(* Schneider Machine Expert - Basic project DDEF, file version 2.7.0.0 *)
(* ProjectInformations: Name=Novo projeto *)

HARDWARE
  Cpu 0: TM221CE24R
  EthernetConfiguration: NetworkName=M221, IpAllocationMode=FixedAddress, IpAddress=0.0.0.0, SubnetMask=0.0.0.0
  SerialLineConfiguration: Baud=Baud19200, Parity=ParityEven, DataBits=DataBits8, StopBits=StopBits1, PhysicalMedium=PhysicalMediumRs485, TransmissionMode=TransmissionModeModbusRtu, SlaveId=1, Addressing=SlaveAddressing
  MastTask: UsePeriodScanMode=false, PeriodScan=100
  FastTask: Period=255
  CpuBehavior: StartingMode=StartAsPreviousState, AutoSaveRamOnEeprom=true, WatchdogPeriod=250

SYMBOLS  (address, symbol, comment, settings)
  %M0       START_
  %M1       STOP
  %M2       RESET
  %M3       EMERGENCIA
  %M4       MANUAL
  %M5       AUTO
  %M6       L_START
  %M7       L_RESET
  %M8       L_STOP
  %M9       L_MANUAL
  %M10      L_AUTO
  %MW0      SNIVEL
  %MW1      SETPOINT
  %MW2      V_ENCHE
  %MW3      V_DESCARGA
  %MW4      V_SETPOINT
  %MW5      V_NIVEL

POU Novo POU
  (* SectionNumber=1 *)

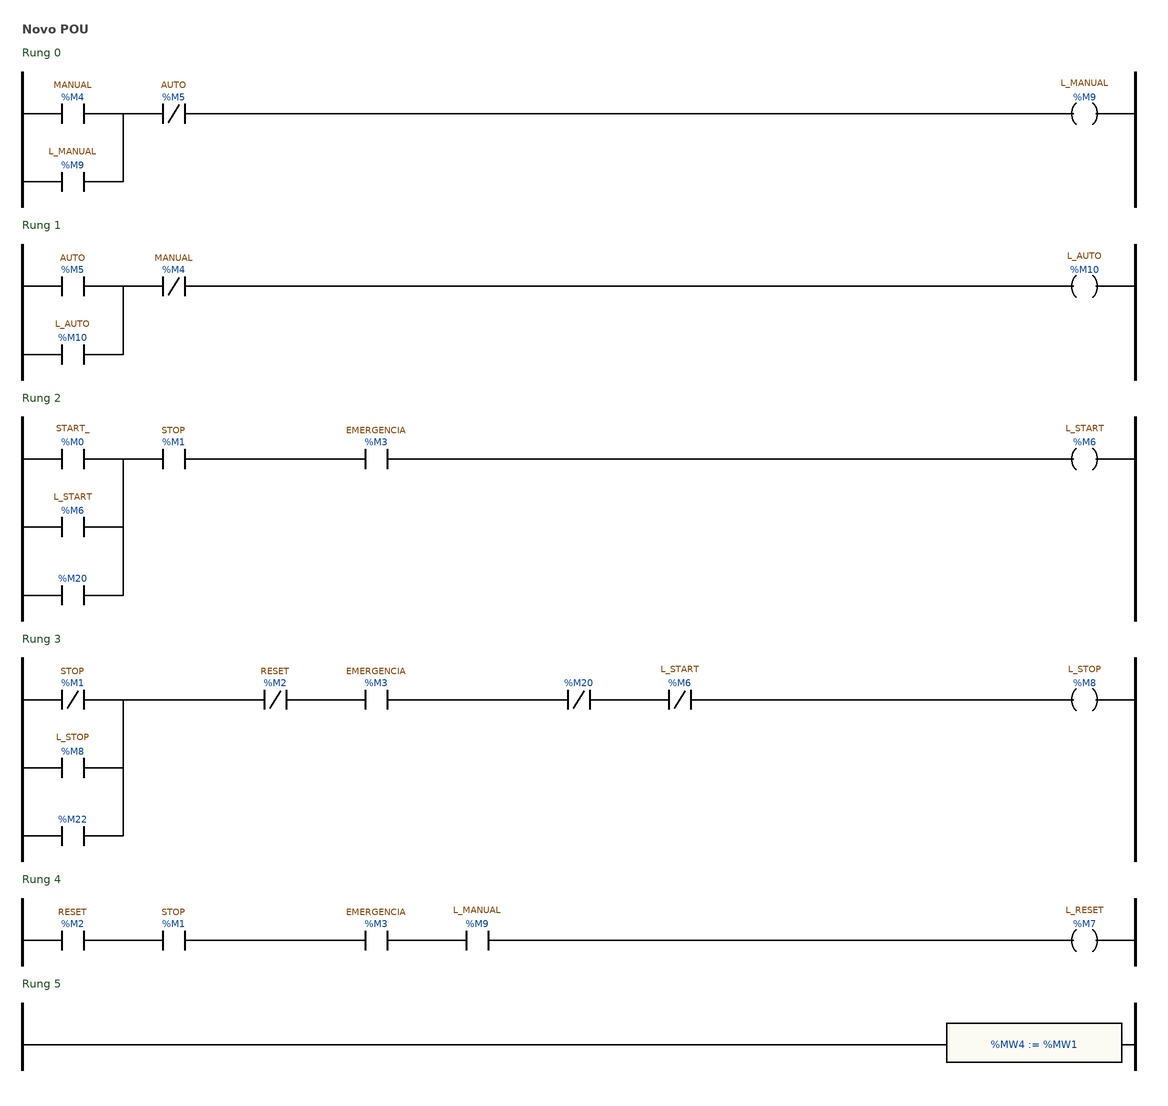

// Rung 0
  LD %M4                  (* MANUAL *)
  OR %M9                  (* L_MANUAL *)
  ANDN %M5                (* AUTO *)
  ST %M9                  (* L_MANUAL *)
  // as ST:
  //   L_MANUAL := (MANUAL OR L_MANUAL) AND NOT AUTO;

// Rung 1
  LD %M5                  (* AUTO *)
  OR %M10                 (* L_AUTO *)
  ANDN %M4                (* MANUAL *)
  ST %M10                 (* L_AUTO *)
  // as ST:
  //   L_AUTO := (AUTO OR L_AUTO) AND NOT MANUAL;

// Rung 2
  LD %M0                  (* START_ *)
  OR %M6                  (* L_START *)
  OR %M20
  AND %M1                 (* STOP *)
  AND %M3                 (* EMERGENCIA *)
  ST %M6                  (* L_START *)
  // as ST:
  //   L_START := (START_ OR L_START OR %M20) AND STOP AND EMERGENCIA;

// Rung 3
  LDN %M1                 (* STOP *)
  OR %M8                  (* L_STOP *)
  OR %M22
  ANDN %M2                (* RESET *)
  AND %M3                 (* EMERGENCIA *)
  ANDN %M20
  ANDN %M6                (* L_START *)
  ST %M8                  (* L_STOP *)
  // as ST:
  //   L_STOP := (NOT STOP OR L_STOP OR %M22) AND NOT RESET AND EMERGENCIA AND NOT %M20 AND NOT L_START;

// Rung 4
  LD %M2                  (* RESET *)
  AND %M1                 (* STOP *)
  AND %M3                 (* EMERGENCIA *)
  AND %M9                 (* L_MANUAL *)
  ST %M7                  (* L_RESET *)
  // as ST:
  //   L_RESET := RESET AND STOP AND EMERGENCIA AND L_MANUAL;

// Rung 5
  LD 1
  [ %MW4 := %MW1 ]        (* V_SETPOINT, SETPOINT *)
  // as ST:
  //   V_SETPOINT := SETPOINT;

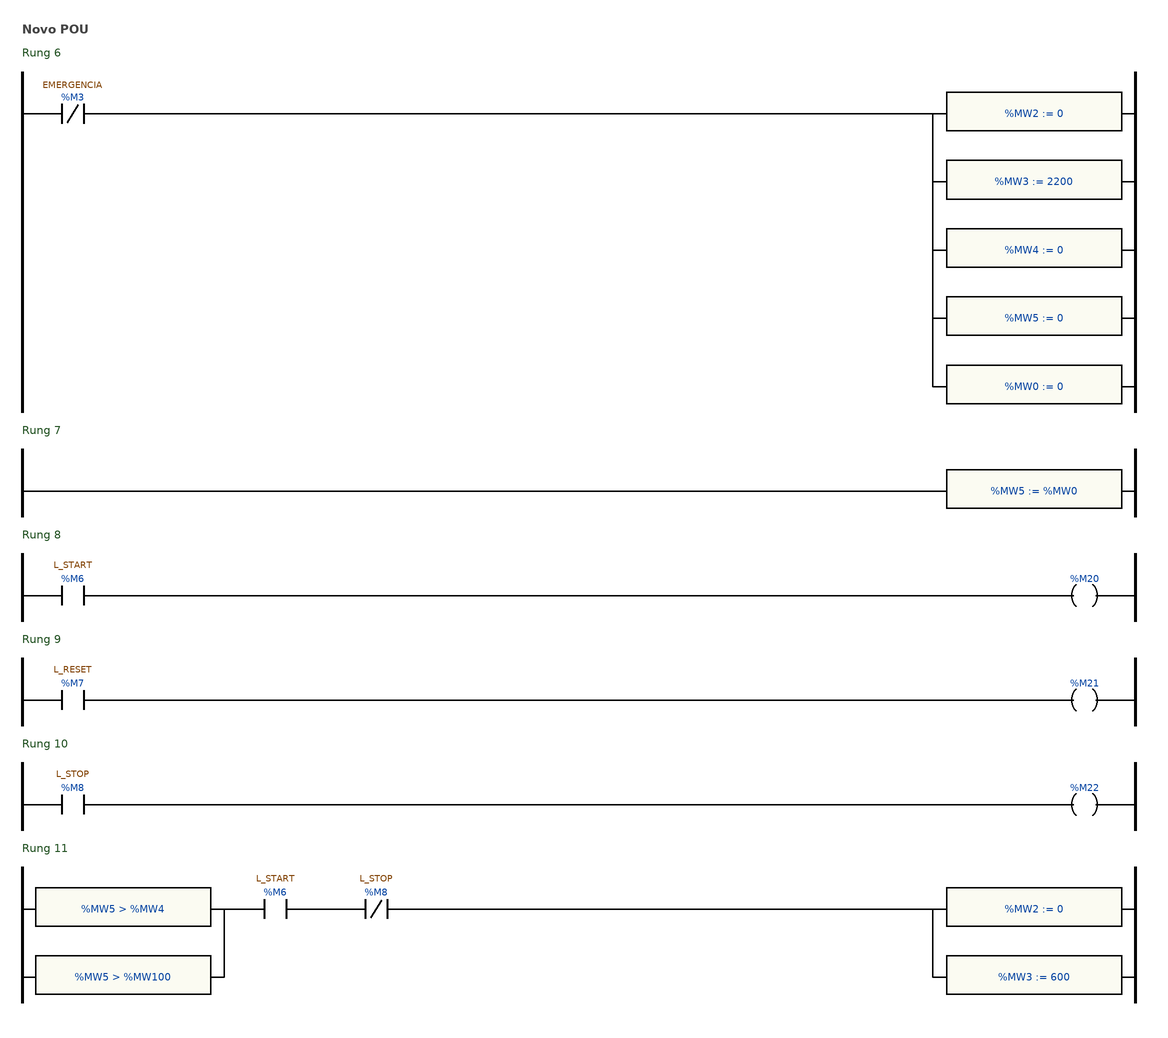

// Rung 6
  LDN %M3                 (* EMERGENCIA *)
  [ %MW2 := 0 ]           (* V_ENCHE *)
  [ %MW3 := 2200 ]        (* V_DESCARGA *)
  [ %MW4 := 0 ]           (* V_SETPOINT *)
  [ %MW5 := 0 ]           (* V_NIVEL *)
  [ %MW0 := 0 ]           (* SNIVEL *)
  // as ST:
  //   IF NOT EMERGENCIA THEN V_ENCHE := 0; END_IF;
  //   IF NOT EMERGENCIA THEN V_DESCARGA := 2200; END_IF;
  //   IF NOT EMERGENCIA THEN V_SETPOINT := 0; END_IF;
  //   IF NOT EMERGENCIA THEN V_NIVEL := 0; END_IF;
  //   IF NOT EMERGENCIA THEN SNIVEL := 0; END_IF;

// Rung 7
  LD 1
  [ %MW5 := %MW0 ]        (* V_NIVEL, SNIVEL *)
  // as ST:
  //   V_NIVEL := SNIVEL;

// Rung 8
  LD %M6                  (* L_START *)
  ST %M20
  // as ST:
  //   %M20 := L_START;

// Rung 9
  LD %M7                  (* L_RESET *)
  ST %M21
  // as ST:
  //   %M21 := L_RESET;

// Rung 10
  LD %M8                  (* L_STOP *)
  ST %M22
  // as ST:
  //   %M22 := L_STOP;

// Rung 11
  LD [ %MW5 > %MW4 ]      (* V_NIVEL, V_SETPOINT *)
  OR [ %MW5 > %MW100 ]    (* V_NIVEL *)
  AND %M6                 (* L_START *)
  ANDN %M8                (* L_STOP *)
  [ %MW2 := 0 ]           (* V_ENCHE *)
  [ %MW3 := 600 ]         (* V_DESCARGA *)
  // as ST:
  //   IF (V_NIVEL > V_SETPOINT OR V_NIVEL > %MW100) AND L_START AND NOT L_STOP THEN V_ENCHE := 0; END_IF;
  //   IF (V_NIVEL > V_SETPOINT OR V_NIVEL > %MW100) AND L_START AND NOT L_STOP THEN V_DESCARGA := 600; END_IF;

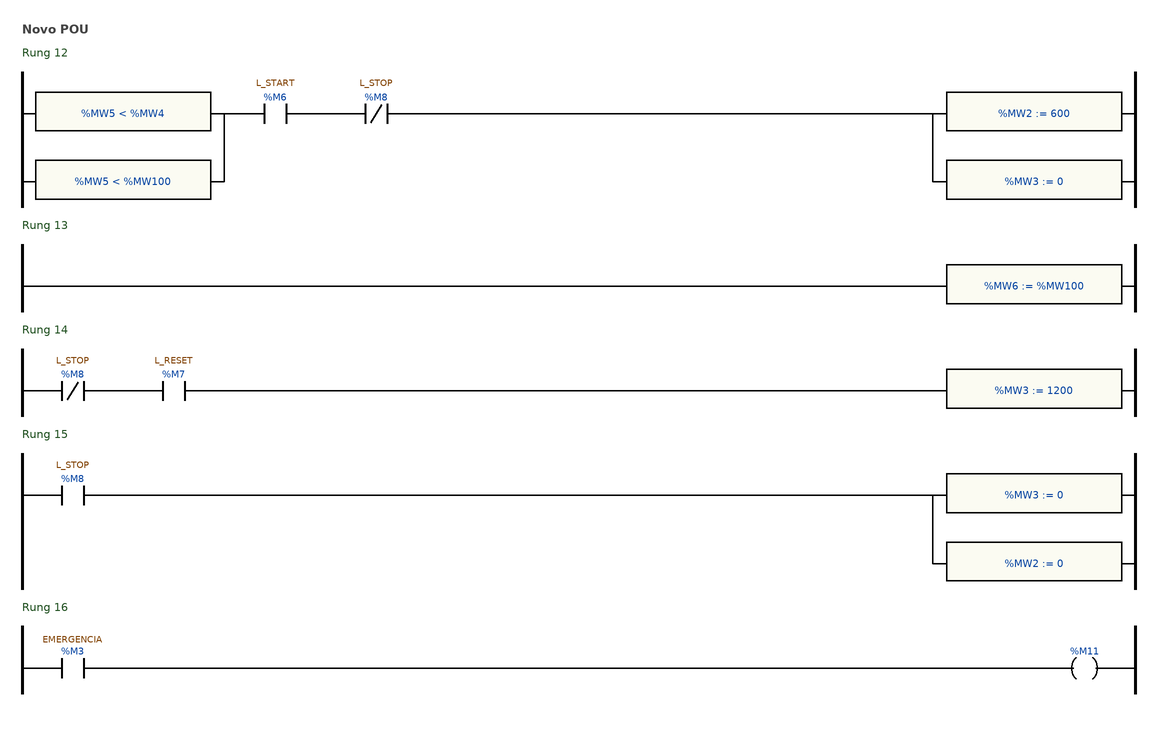

// Rung 12
  LD [ %MW5 < %MW4 ]      (* V_NIVEL, V_SETPOINT *)
  OR [ %MW5 < %MW100 ]    (* V_NIVEL *)
  AND %M6                 (* L_START *)
  ANDN %M8                (* L_STOP *)
  [ %MW2 := 600 ]         (* V_ENCHE *)
  [ %MW3 := 0 ]           (* V_DESCARGA *)
  // as ST:
  //   IF (V_NIVEL < V_SETPOINT OR V_NIVEL < %MW100) AND L_START AND NOT L_STOP THEN V_ENCHE := 600; END_IF;
  //   IF (V_NIVEL < V_SETPOINT OR V_NIVEL < %MW100) AND L_START AND NOT L_STOP THEN V_DESCARGA := 0; END_IF;

// Rung 13
  LD 1
  [ %MW6 := %MW100 ]
  // as ST:
  //   %MW6 := %MW100;

// Rung 14
  LDN %M8                 (* L_STOP *)
  AND %M7                 (* L_RESET *)
  [ %MW3 := 1200 ]        (* V_DESCARGA *)
  // as ST:
  //   IF NOT L_STOP AND L_RESET THEN V_DESCARGA := 1200; END_IF;

// Rung 15
  LD %M8                  (* L_STOP *)
  [ %MW3 := 0 ]           (* V_DESCARGA *)
  [ %MW2 := 0 ]           (* V_ENCHE *)
  // as ST:
  //   IF L_STOP THEN V_DESCARGA := 0; END_IF;
  //   IF L_STOP THEN V_ENCHE := 0; END_IF;

// Rung 16
  LD %M3                  (* EMERGENCIA *)
  ST %M11
  // as ST:
  //   %M11 := EMERGENCIA;
